FUNCTION_BLOCK FB_CalcFocalLengthSingleLens EXTENDS FB_Fallible IMPLEMENTS I_CalcFocalLengthSingleLens
VAR
    iCalcXRayDelta : I_CalcXRayDelta; // The x-ray delta, the real part of the index of refraction, unitless value.

    {attribute 'pytmc' := '
        pv: FocalLength
        io: i
        field: DESC Calculated focal length of lens.
    '}
    fFocalLength : LREAL; // The focal length of the lens.
END_VAR


METHOD Calculate : LREAL
VAR_INPUT
    iLens : I_Lens;
END_VAR
VAR
    fDelta : LREAL;
END_VAR

// Initialize focal length and error values.
fFocalLength := 0.0;
ClearError();

// Check for an invalid lens input.
IF iLens.GetError() THEN
    SetError(
        sMsg := CONCAT('The input lens has the following error message: [',
        CONCAT(iLens.GetErrorMsg(),
        ']'))
    );
    RETURN;
END_IF

fDelta := iCalcXRayDelta.Calculate(sChemicalFormula := iLens.MaterialName);

// Check for an invalid delta input.
IF iCalcXRayDelta.GetError() THEN
    SetError(
        sMsg := CONCAT('The input delta has the following error message: [',
        CONCAT(iCalcXRayDelta.GetErrorMsg(),
        ']'))
    );
    RETURN;
END_IF

IF fDelta = 0.0 THEN
    SetError(
        sMsg := CONCAT('The delta calculated: [',
        CONCAT(LREAL_TO_STRING(fDelta),
        '] must not be 0.'))
    );
    RETURN;
END_IF

IF iLens.Radius <= 0.0 THEN
    SetError(
        sMsg := CONCAT('The radius specified: [',
        CONCAT(LREAL_TO_STRING(iLens.Radius),
        '] must be greater than 0.'))
    );
    RETURN;
END_IF

fFocalLength := iLens.Radius / 2.0 / fDelta;

Calculate := fFocalLength;
END_METHOD


METHOD FB_init : BOOL
VAR_INPUT
    bInitRetains : BOOL; // if TRUE, the retain variables are initialized (warm start / cold start)
    bInCopyCode : BOOL;  // if TRUE, the instance afterwards gets moved into the copy code (online change)

    iCalcXRayDelta : I_CalcXRayDelta; // The x-ray delta, the real part of the index of refraction, unitless value.
END_VAR

THIS^.iCalcXRayDelta := iCalcXRayDelta;
END_METHOD

END_FUNCTION_BLOCK

(* stored: Version 1.1.0.1
   POU FB_CalcFocalLengthSingleLens: Id {4986d52d-63ec-4366-87a7-ec07b5c7c44d}, SpecialFunc None
   Method Calculate: Id {ccac877d-2b8a-4013-bf1b-351f6a9d80e6}
   Method FB_init: Id {20bb0204-195a-417d-97fe-efa1e33a672d} *)
